(* IEC 61131-3 sources: eCockpitGit/test_project/src/%F%00 Library/%F%Structured Buffer Read Write Base/%ITF%ITF_StructReaderBase/%F%Structure, 6 files *)

(* ---- %METH%compareKeyName.st ---- *)
//This method compares a string to the selected string
METHOD compareKeyName : EStructType
VAR_INPUT
	name				:POINTER TO EASCII;
END_VAR
(*%!%__DELIMITER__%!%*)

(* ---- %METH%exportSelection.st ---- *)
//This method returns the buffer position and size of the currently selected struct/object
METHOD exportSelection : BOOL
VAR_OUTPUT
	position		:POINTER TO EASCII;
	size			:DWORD;
END_VAR
(*%!%__DELIMITER__%!%*)

(* ---- %METH%findKey.st ---- *)
//This method finds a key by name in the selected structure
METHOD findKey : EStructType
VAR_INPUT
	name			:POINTER TO EASCII;		//Address of the name to find, only input string address or zero terminated byte array
END_VAR

(*%!%__DELIMITER__%!%*)

(* ---- %METH%readKeyName.st ---- *)
//This method returns the name of the currently selected key
//Returns true on output if value is valid
METHOD readKeyName : BOOL
VAR_INPUT
	name			:POINTER TO EASCII;		//Address of the name to find, only input string address or zero terminated byte array
	lenMax			:DWORD;					//Max lenght of string value
END_VAR
VAR_OUTPUT
	len				:WORD;					//Actual lenght of string value
END_VAR
(*%!%__DELIMITER__%!%*)

(* ---- %METH%readKeyNameChar.st ---- *)
//This method returns the character of a given position from the key name
//Returns null if out of range
//1 is the first character, 0 is also the first character
METHOD readKeyNameChar : EASCII
VAR_INPUT
	charNum			:WORD;		//Character number
END_VAR

(*%!%__DELIMITER__%!%*)

(* ---- %METH%readKeyNameLevel.st ---- *)
//This method returns the name of a specific level in the struct
//Returns true on output if value is valid
METHOD readKeyNameLevel : BOOL
VAR_INPUT
	name			:POINTER TO EASCII;		//Address of the name to find, only input string address or zero terminated byte array
	lenMax			:DWORD;					//Max lenght of string value
	level			:BYTE;					//The level to get from
END_VAR
VAR_OUTPUT
	len				:WORD;					//Actual lenght of string value
END_VAR
(*%!%__DELIMITER__%!%*)
